SYSTEM ModSFunctions
  (* Version 1.0, Author, 4DIAC-Consortium *)
  APPLICATION Constants
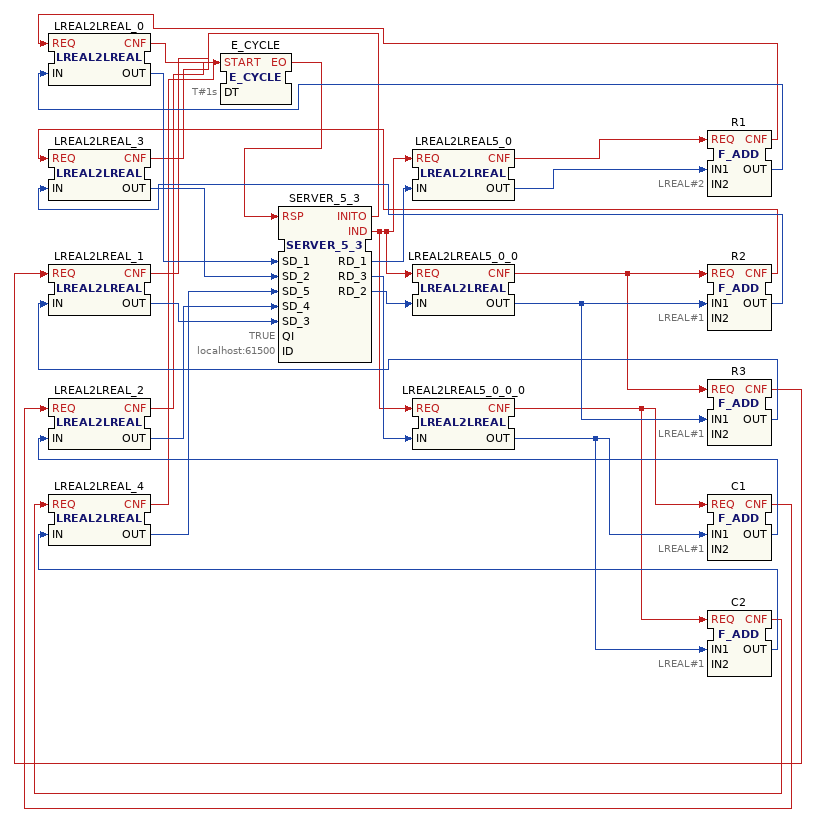
    FBS
      LREAL2LREAL_0 : LREAL2LREAL;
      LREAL2LREAL_3 : LREAL2LREAL;
      E_CYCLE : E_CYCLE(DT := T#1s);
      SERVER_5_3 : SERVER_5_3(QI := TRUE, ID := localhost:61500);
      LREAL2LREAL_1 : LREAL2LREAL;
      LREAL2LREAL_4 : LREAL2LREAL;
      LREAL2LREAL_2 : LREAL2LREAL;
      LREAL2LREAL5_0 : LREAL2LREAL;
      LREAL2LREAL5_0_0_0 : LREAL2LREAL;
      LREAL2LREAL5_0_0 : LREAL2LREAL;
      R1 : F_ADD(IN2 := LREAL#2);
      R2 : F_ADD(IN2 := LREAL#1);
      R3 : F_ADD(IN2 := LREAL#1);
      C2 : F_ADD(IN2 := LREAL#1);
      C1 : F_ADD(IN2 := LREAL#1);
    END_FBS
    EVENT_CONNECTIONS
      LREAL2LREAL_0.CNF TO E_CYCLE.START;
      LREAL2LREAL_3.CNF TO E_CYCLE.START;
      SERVER_5_3.INITO TO E_CYCLE.START;
      E_CYCLE.EO TO SERVER_5_3.RSP;
      LREAL2LREAL_1.CNF TO E_CYCLE.START;
      LREAL2LREAL_2.CNF TO E_CYCLE.START;
      LREAL2LREAL_4.CNF TO E_CYCLE.START;
      SERVER_5_3.IND TO LREAL2LREAL5_0.REQ;
      SERVER_5_3.IND TO LREAL2LREAL5_0_0_0.REQ;
      SERVER_5_3.IND TO LREAL2LREAL5_0_0.REQ;
      LREAL2LREAL5_0.CNF TO R1.REQ;
      R1.CNF TO LREAL2LREAL_0.REQ;
      LREAL2LREAL5_0_0.CNF TO R2.REQ;
      R2.CNF TO LREAL2LREAL_3.REQ;
      LREAL2LREAL5_0_0.CNF TO R3.REQ;
      R3.CNF TO LREAL2LREAL_1.REQ;
      LREAL2LREAL5_0_0_0.CNF TO C2.REQ;
      C2.CNF TO LREAL2LREAL_4.REQ;
      LREAL2LREAL5_0_0_0.CNF TO C1.REQ;
      C1.CNF TO LREAL2LREAL_2.REQ;
    END_CONNECTIONS
    DATA_CONNECTIONS
      LREAL2LREAL_0.OUT TO SERVER_5_3.SD_1;
      LREAL2LREAL_3.OUT TO SERVER_5_3.SD_2;
      LREAL2LREAL_4.OUT TO SERVER_5_3.SD_5;
      LREAL2LREAL_2.OUT TO SERVER_5_3.SD_4;
      LREAL2LREAL_1.OUT TO SERVER_5_3.SD_3;
      SERVER_5_3.RD_1 TO LREAL2LREAL5_0.IN;
      SERVER_5_3.RD_3 TO LREAL2LREAL5_0_0_0.IN;
      SERVER_5_3.RD_2 TO LREAL2LREAL5_0_0.IN;
      LREAL2LREAL5_0.OUT TO R1.IN1;
      R1.OUT TO LREAL2LREAL_0.IN;
      LREAL2LREAL5_0_0.OUT TO R2.IN1;
      R2.OUT TO LREAL2LREAL_3.IN;
      LREAL2LREAL5_0_0.OUT TO R3.IN1;
      R3.OUT TO LREAL2LREAL_1.IN;
      LREAL2LREAL5_0_0_0.OUT TO C2.IN1;
      C2.OUT TO LREAL2LREAL_4.IN;
      LREAL2LREAL5_0_0_0.OUT TO C1.IN1;
      C1.OUT TO LREAL2LREAL_2.IN;
    END_CONNECTIONS
  END_APPLICATION
  APPLICATION aa
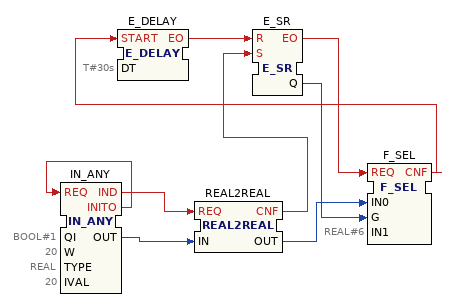
    FBS
      E_SR : E_SR;
      E_DELAY : E_DELAY(DT := T#30s);
      F_SEL : F_SEL(IN1 := REAL#6);
      REAL2REAL : REAL2REAL;
      IN_ANY : IN_ANY(QI := BOOL#1, W := 20, TYPE := REAL, IVAL := 20);
    END_FBS
    EVENT_CONNECTIONS
      E_DELAY.EO TO E_SR.R;
      E_SR.EO TO F_SEL.REQ;
      REAL2REAL.CNF TO E_SR.S;
      F_SEL.CNF TO E_DELAY.START;
      IN_ANY.IND TO REAL2REAL.REQ;
      IN_ANY.INITO TO IN_ANY.REQ;
    END_CONNECTIONS
    DATA_CONNECTIONS
      REAL2REAL.OUT TO F_SEL.IN0;
      E_SR.Q TO F_SEL.G;
      IN_ANY.OUT TO REAL2REAL.IN;
    END_CONNECTIONS
  END_APPLICATION
  DEVICE FORTE_PC : FORTE_PC(MGR_ID := "localhost:61500")
    {SET_ATTRIBUTE(Profile, HOLOBLOC)}
    RESOURCE EMB_RES : EMB_RES
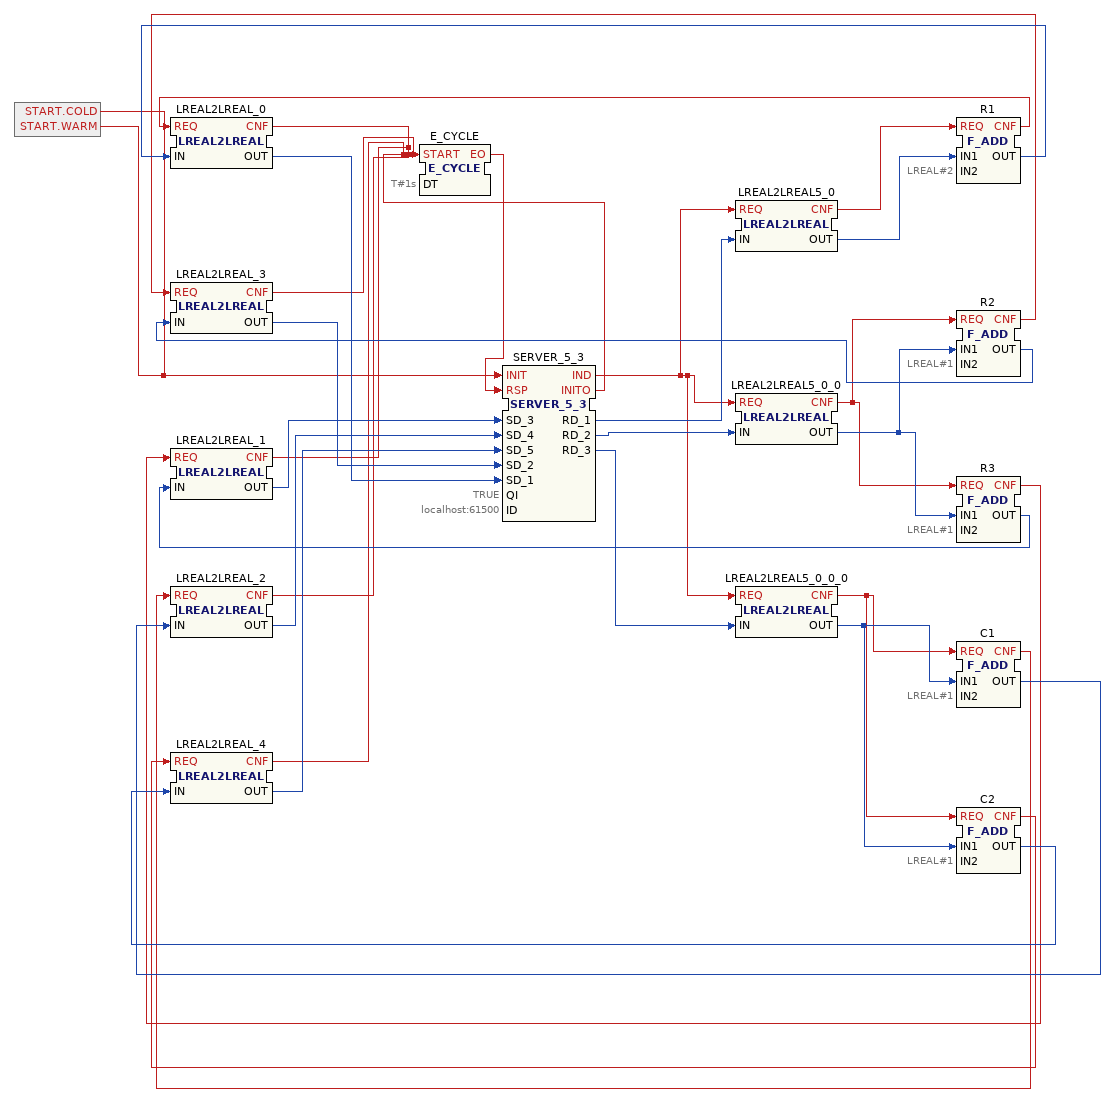
      FBS
        C1 : F_ADD(IN2 := LREAL#1);
        C2 : F_ADD(IN2 := LREAL#1);
        R3 : F_ADD(IN2 := LREAL#1);
        R2 : F_ADD(IN2 := LREAL#1);
        R1 : F_ADD(IN2 := LREAL#2);
        LREAL2LREAL5_0_0 : LREAL2LREAL;
        LREAL2LREAL5_0_0_0 : LREAL2LREAL;
        LREAL2LREAL5_0 : LREAL2LREAL;
        LREAL2LREAL_2 : LREAL2LREAL;
        LREAL2LREAL_4 : LREAL2LREAL;
        LREAL2LREAL_1 : LREAL2LREAL;
        SERVER_5_3 : SERVER_5_3(QI := TRUE, ID := localhost:61500);
        E_CYCLE : E_CYCLE(DT := T#1s);
        LREAL2LREAL_3 : LREAL2LREAL;
        LREAL2LREAL_0 : LREAL2LREAL;
      END_FBS
      EVENT_CONNECTIONS
        LREAL2LREAL5_0_0.CNF TO R2.REQ;
        LREAL2LREAL5_0_0.CNF TO R3.REQ;
        LREAL2LREAL5_0_0_0.CNF TO C2.REQ;
        LREAL2LREAL5_0_0_0.CNF TO C1.REQ;
        LREAL2LREAL5_0.CNF TO R1.REQ;
        C1.CNF TO LREAL2LREAL_2.REQ;
        C2.CNF TO LREAL2LREAL_4.REQ;
        R3.CNF TO LREAL2LREAL_1.REQ;
        START.COLD TO SERVER_5_3.INIT;
        START.WARM TO SERVER_5_3.INIT;
        SERVER_5_3.IND TO LREAL2LREAL5_0.REQ;
        SERVER_5_3.IND TO LREAL2LREAL5_0_0_0.REQ;
        SERVER_5_3.IND TO LREAL2LREAL5_0_0.REQ;
        SERVER_5_3.INITO TO E_CYCLE.START;
        LREAL2LREAL_1.CNF TO E_CYCLE.START;
        LREAL2LREAL_2.CNF TO E_CYCLE.START;
        LREAL2LREAL_4.CNF TO E_CYCLE.START;
        E_CYCLE.EO TO SERVER_5_3.RSP;
        R2.CNF TO LREAL2LREAL_3.REQ;
        LREAL2LREAL_3.CNF TO E_CYCLE.START;
        R1.CNF TO LREAL2LREAL_0.REQ;
        LREAL2LREAL_0.CNF TO E_CYCLE.START;
      END_CONNECTIONS
      DATA_CONNECTIONS
        LREAL2LREAL5_0_0.OUT TO R2.IN1;
        LREAL2LREAL5_0_0.OUT TO R3.IN1;
        LREAL2LREAL5_0_0_0.OUT TO C2.IN1;
        LREAL2LREAL5_0_0_0.OUT TO C1.IN1;
        LREAL2LREAL5_0.OUT TO R1.IN1;
        C1.OUT TO LREAL2LREAL_2.IN;
        C2.OUT TO LREAL2LREAL_4.IN;
        R3.OUT TO LREAL2LREAL_1.IN;
        LREAL2LREAL_1.OUT TO SERVER_5_3.SD_3;
        LREAL2LREAL_2.OUT TO SERVER_5_3.SD_4;
        LREAL2LREAL_4.OUT TO SERVER_5_3.SD_5;
        SERVER_5_3.RD_1 TO LREAL2LREAL5_0.IN;
        SERVER_5_3.RD_2 TO LREAL2LREAL5_0_0.IN;
        SERVER_5_3.RD_3 TO LREAL2LREAL5_0_0_0.IN;
        R2.OUT TO LREAL2LREAL_3.IN;
        LREAL2LREAL_3.OUT TO SERVER_5_3.SD_2;
        R1.OUT TO LREAL2LREAL_0.IN;
        LREAL2LREAL_0.OUT TO SERVER_5_3.SD_1;
      END_CONNECTIONS
    END_RESOURCE
  END_DEVICE
  DEVICE FORTE_PC_1 : FORTE_PC(MGR_ID := "localhost:61499")
    {SET_ATTRIBUTE(Profile, HOLOBLOC)}
    RESOURCE EMB_RES : EMB_RES
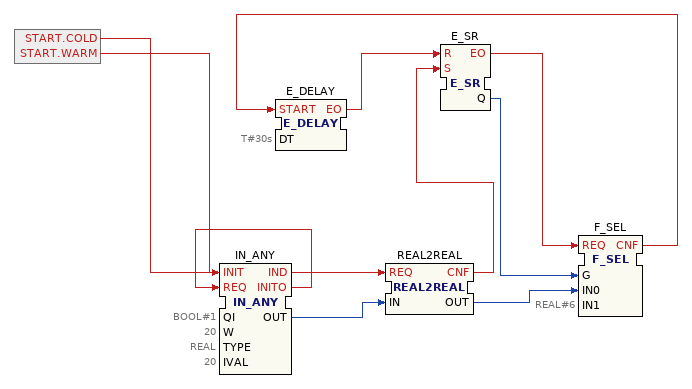
      FBS
        E_DELAY : E_DELAY(DT := T#30s);
        E_SR : E_SR;
        REAL2REAL : REAL2REAL;
        IN_ANY : IN_ANY(QI := BOOL#1, W := 20, TYPE := REAL, IVAL := 20);
        F_SEL : F_SEL(IN1 := REAL#6);
      END_FBS
      EVENT_CONNECTIONS
        E_DELAY.EO TO E_SR.R;
        REAL2REAL.CNF TO E_SR.S;
        IN_ANY.IND TO REAL2REAL.REQ;
        E_SR.EO TO F_SEL.REQ;
        F_SEL.CNF TO E_DELAY.START;
        START.COLD TO IN_ANY.INIT;
        START.WARM TO IN_ANY.INIT;
        IN_ANY.INITO TO IN_ANY.REQ;
      END_CONNECTIONS
      DATA_CONNECTIONS
        IN_ANY.OUT TO REAL2REAL.IN;
        E_SR.Q TO F_SEL.G;
        REAL2REAL.OUT TO F_SEL.IN0;
      END_CONNECTIONS
    END_RESOURCE
  END_DEVICE
  MAPPINGS
    Constants.LREAL2LREAL_0 ON FORTE_PC.EMB_RES.LREAL2LREAL_0;
    Constants.LREAL2LREAL_3 ON FORTE_PC.EMB_RES.LREAL2LREAL_3;
    Constants.E_CYCLE ON FORTE_PC.EMB_RES.E_CYCLE;
    Constants.SERVER_5_3 ON FORTE_PC.EMB_RES.SERVER_5_3;
    Constants.LREAL2LREAL_1 ON FORTE_PC.EMB_RES.LREAL2LREAL_1;
    Constants.LREAL2LREAL_4 ON FORTE_PC.EMB_RES.LREAL2LREAL_4;
    Constants.LREAL2LREAL_2 ON FORTE_PC.EMB_RES.LREAL2LREAL_2;
    Constants.LREAL2LREAL5_0 ON FORTE_PC.EMB_RES.LREAL2LREAL5_0;
    Constants.LREAL2LREAL5_0_0_0 ON FORTE_PC.EMB_RES.LREAL2LREAL5_0_0_0;
    Constants.LREAL2LREAL5_0_0 ON FORTE_PC.EMB_RES.LREAL2LREAL5_0_0;
    Constants.R1 ON FORTE_PC.EMB_RES.R1;
    Constants.R2 ON FORTE_PC.EMB_RES.R2;
    Constants.R3 ON FORTE_PC.EMB_RES.R3;
    Constants.C2 ON FORTE_PC.EMB_RES.C2;
    Constants.C1 ON FORTE_PC.EMB_RES.C1;
    aa.E_SR ON FORTE_PC_1.EMB_RES.E_SR;
    aa.E_DELAY ON FORTE_PC_1.EMB_RES.E_DELAY;
    aa.F_SEL ON FORTE_PC_1.EMB_RES.F_SEL;
    aa.REAL2REAL ON FORTE_PC_1.EMB_RES.REAL2REAL;
    aa.IN_ANY ON FORTE_PC_1.EMB_RES.IN_ANY;
  END_MAPPINGS
  SEGMENTS
    Ethernet : Ethernet;
  END_SEGMENTS
  LINKS
    FORTE_PC_1 => Ethernet;
  END_LINKS
END_SYSTEM
